FUNCTION_BLOCK FbDeadBand (* Зона нечувствительности. *)
  (* Standard: 61499-1; Description: Зона нечувствительности. Simple FB with one algorithm *)
  (* Version 2.2, 2026-03-20, VA, LIB_PLC *)
  (* Documentation:
  // Зона нечувствительности. //      DbDeadBand //    +------------+ //    | FbDeadBand | // ->-|In       Out|->- //   -|ERMAX       | //   -|ERMIN       | //    +------------+ // Условное графическое обозначение. // //          ERMAX //      +-----------+ //      |           | //      |       /   | //      |      /    | //      |      |    | // In->-|   +--+    |->-Out //      |   |       | //      |  /        | //      | /         | //      |           | //      +-----------+ //          ERMIN // Статическая характеристика. // //                +Out //                  |        * //                  |       * //                  |      * //                  |     * //                  |     * //                  |     * //             ERMIN|     * //            |<--->|     * //            |     |     * // -In <------*************--> +In //            *     |     | //            *     |<--->| //            *     |ERMAX //            *     | //            *     | //            *     | //           *      | //          *       | //         *        | //                -Out // Временная характеристика. // // +In // |            * // |           * * // |----------*---* ----------------- // |         *     *               | // |        *       *              | ERMAX // |       *         *             | // +------*-----------*----------------------> t[s] // |     *             *           | // |    *               *          | ERMIN // |   *                 *         | // |--*-------------------*---------- // | *                     * // |*                       * // -In // // +Out // |            * // |           * * // |----------*---* ----------------- // |          *   *                | // |          *   *                | ERMAX // |          *   *                | // +--*********---*********------------------> t[s] // |  *                   *        | // |  *                   *        | ERMIN // |  *                   *        | // |--*-------------------*---------- // | *                     * // |*                       * // -Out
  *)
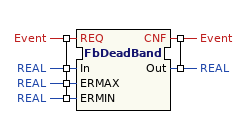
  EVENT_INPUT
    REQ WITH In, ERMAX, ERMIN; (* Normal Execution Request *)
  END_EVENT
  EVENT_OUTPUT
    CNF WITH Out; (* Execution Confirmation *)
  END_EVENT
  VAR_INPUT
    In : REAL := 0.0; (* Вход зоны нечувствительности. *)
    ERMAX : REAL := 0.001; (* Зона нечувствительности верхняя граница. *)
    ERMIN : REAL := -0.001; (* Зона нечувствительности нижняя граница. *)
  END_VAR
  VAR_OUTPUT
    Out : REAL := 0.0; (* Выход зоны нечувствительности. *)
  END_VAR
  EC_STATES
    REQ : REQ -> CNF;
  END_STATES
  ALGORITHM REQ IN ST:
// Зона нечувствительности.
IF ((ERMIN < In) AND (In < ERMAX)) THEN
	Out := 0.0;
ELSE
	Out := In;
END_IF;

// @COPYLEFT ALL WRONGS RESERVED :)
// Author: VA
// Contacts: DIY.PLC.314@gmail.com
// Date start LIB_PLC: 2014
// License: GNU GPL-2.0-or-later
// https://www.gnu.org/licenses/old-licenses/gpl-2.0.html
// https://www.youtube.com/watch?v=n1F_MfLRlX0
// https://www.youtube.com/@DIY_PLC
// https://github.com/DIYPLC/LIB_PLC
// https://oshwlab.com/diy.plc.314/PLC_HW1_SW1
// https://3dtoday.ru/3d-models/mechanical-parts/body/korpus-na-din-reiku
// https://t.me/DIY_PLC
  END_ALGORITHM
END_FUNCTION_BLOCK
